// TIA Portal project "start stop" (V16)

(* hardware
DEVICE "S7-1200 station_1"  S7-1200 Station
   slot 0: "Rack_0"  S7-1200 Rack  Rack  V1.0
   slot 1: "PLC_1"  CPU 1212C AC/DC/Rly  6ES7 212-1BE40-0XB0  V4.0
*)

// ===== PLC "PLC_1"  CPU 1212C AC/DC/Rly =====

VAR_GLOBAL   // PLC tag table "Default tag table"
   "start" AT %I0.2 : Bool;
   "K1" AT %Q0.0 : Bool;
   "stop1" AT %I0.4 : Bool;
   "k2" AT %Q0.1 : Bool;
   "start2" AT %I0.3 : Bool;
   "T1 tag" AT %M0.0 : Bool;
   "RTU2 tag" AT %M0.1 : Bool;
   "X" AT %M0.2 : Bool;
   "C1 tag" AT %M0.3 : Bool;
   "k1 tag" AT %M0.4 : Bool;
   "RTU1 tag" AT %M0.6 : Bool;
   "Tag_1" AT %M0.7 : Bool;
   "k3" AT %Q0.2 : Bool;
   "Tag_2" AT %M0.5 : Bool;
END_VAR

// folder: System blocks/Program resources

DATA_BLOCK "RTU1"   // DB1
{ S7_Optimized_Access := 'TRUE' }
AUTHOR : Simatic
FAMILY : IEC
NAME : IEC_TMR
VERSION : 1.0
// stored: InstanceOfName IEC_TIMER
"IEC_TIMER"
BEGIN
END_DATA_BLOCK

// folder: (top level)

ORGANIZATION_BLOCK "Main"   // OB1, LAD, ProgramCycle
TITLE = "Main Program Sweep (Cycle)"
{ S7_Optimized_Access := 'TRUE' }
VERSION : 0.1
   VAR_INPUT
      Initial_Call : Bool;   // Initial call of this OB
      Remanence : Bool;   // =True, if remanent data are available
   END_VAR
BEGIN

REGION Network 1
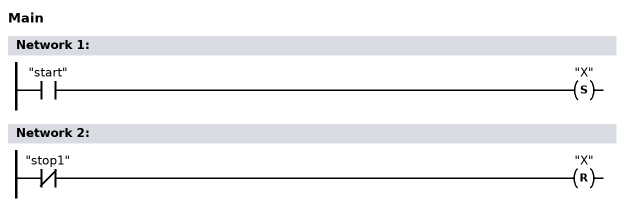
   RUNG wire#powerrail
      Contact( "start" )
      S_Coil( "X" )
   END_RUNG
   // the same network as SCL:
   IF "start" THEN "X" := TRUE; END_IF;
END_REGION

REGION Network 2
   RUNG wire#powerrail
      I_Contact( "stop1" )
      R_Coil( "X" )
   END_RUNG
   // the same network as SCL:
   IF NOT "stop1" THEN "X" := FALSE; END_IF;
END_REGION
END_ORGANIZATION_BLOCK